LIN {X 0,Y 62.695,Z 614.162,A -85,B 0,C 180,E1 -28667.729,E2 -28667.729} C_VEL
LIN {X 0,Y 62.128,Z 611.496,A -85,B 0,C 180,E1 -28675.552,E2 -28675.552} C_VEL
LIN {X 0,Y 62.961,Z 606.814,A -85,B 0,C 180,E1 -28685.536,E2 -28685.536} C_VEL
LIN {X 0,Y 64.666,Z 601.68,A -85,B 0,C 180,E1 -28693.508,E2 -28693.508} C_VEL
LIN {X 0,Y 66.583,Z 596.849,A -85,B 0,C 180,E1 -28699.352,E2 -28699.352} C_VEL
LIN {X 0,Y 69.574,Z 589.721,A -85,B 0,C 180,E1 -28705.944,E2 -28705.944} C_VEL
LIN {X 0,Y 73.049,Z 581.764,A -85,B 0,C 180,E1 -28711.375,E2 -28711.375} C_VEL
LIN {X 0,Y 74.263,Z 578.204,A -85,B 0,C 180,E1 -28713.388,E2 -28713.388} C_VEL
LIN {X 0,Y 75.02,Z 569.916,A -85,B 0,C 180,E1 -28718.075,E2 -28718.075} C_VEL
LIN {X 0,Y 75.368,Z 562.819,A -85,B 0,C 180,E1 -28721.537,E2 -28721.537} C_VEL
LIN {X 0,Y 75.411,Z 557.992,A -85,B 0,C 180,E1 -28723.736,E2 -28723.736} C_VEL
LIN {X 0,Y 75.17,Z 557.115,A -85,B 0,C 180,E1 -28724.205,E2 -28724.205} C_VEL
LIN {X 0,Y 73.982,Z 554.238,A -85,B 0,C 180,E1 -28726.014,E2 -28726.014} C_VEL
LIN {X 0,Y 71.312,Z 550.768,A -85,B 0,C 180,E1 -28729.127,E2 -28729.127} C_VEL
LIN {X 0,Y 68.058,Z 548.078,A -85,B 0,C 180,E1 -28732.584,E2 -28732.584} C_VEL
LIN {X 0,Y 63.467,Z 544.939,A -85,B 0,C 180,E1 -28737.902,E2 -28737.902} C_VEL
LIN {X 0,Y 59.445,Z 541.388,A -85,B 0,C 180,E1 -28743.729,E2 -28743.729} C_VEL
LIN {X 0,Y 58.168,Z 538.724,A -85,B 0,C 180,E1 -28746.42,E2 -28746.42} C_VEL
LIN {X 0,Y 58.056,Z 538.062,A -85,B 0,C 180,E1 -28746.892,E2 -28746.892} C_VEL
LIN {X 0,Y 58.093,Z 538.06,A -85,B 0,C 180,E1 -28756.537,E2 -28756.537} C_VEL
LIN {X 0,Y 58.073,Z 538.046,A -85,B 0,C 180,E1 -28762.763,E2 -28762.763} C_VEL
LIN {X 0,Y 58.154,Z 538.049,A -85,B 0,C 180,E1 -28771.091,E2 -28771.091} C_VEL
LIN {X 0,Y 58.523,Z 538.007,A -85,B 0,C 180,E1 -28783.874,E2 -28783.874} C_VEL
LIN {X 0,Y 58.819,Z 537.971,A -85,B 0,C 180,E1 -28793.137,E2 -28793.137} C_VEL
LIN {X 0,Y 59.394,Z 537.882,A -85,B 0,C 180,E1 -28799.999,E2 -28799.999} C_VEL
LIN {X 0,Y 58.822,Z 537.967,A -85,B 0,C 180,E1 -28806.861,E2 -28806.861} C_VEL
LIN {X 0,Y 58.656,Z 537.992,A -85,B 0,C 180,E1 -28813.864,E2 -28813.864} C_VEL
LIN {X 0,Y 58.313,Z 538.113,A -85,B 0,C 180,E1 -28819.168,E2 -28819.168} C_VEL
LIN {X 0,Y 59.17,Z 540.867,A -85,B 0,C 180,E1 -28821.33,E2 -28821.33} C_VEL
LIN {X 0,Y 61.251,Z 543.062,A -85,B 0,C 180,E1 -28824.578,E2 -28824.578} C_VEL
LIN {X 0,Y 63.526,Z 546.992,A -85,B 0,C 180,E1 -28828.49,E2 -28828.49} C_VEL
LIN {X 0,Y 65.839,Z 551.416,A -85,B 0,C 180,E1 -28832.257,E2 -28832.257} C_VEL
LIN {X 0,Y 67.801,Z 556.21,A -85,B 0,C 180,E1 -28835.78,E2 -28835.78} C_VEL
LIN {X 0,Y 69.602,Z 562.062,A -85,B 0,C 180,E1 -28839.511,E2 -28839.511} C_VEL
LIN {X 0,Y 69.534,Z 564.952,A -85,B 0,C 180,E1 -28840.948,E2 -28840.948} C_VEL
LIN {X 0,Y 68.595,Z 571.827,A -85,B 0,C 180,E1 -28844.181,E2 -28844.181} C_VEL
LIN {X 0,Y 67.006,Z 579.314,A -85,B 0,C 180,E1 -28848.237,E2 -28848.237} C_VEL
LIN {X 0,Y 65.019,Z 587.202,A -85,B 0,C 180,E1 -28853.527,E2 -28853.527} C_VEL
LIN {X 0,Y 61.812,Z 594.337,A -85,B 0,C 180,E1 -28859.23,E2 -28859.23} C_VEL
LIN {X 0,Y 58.654,Z 601.567,A -85,B 0,C 180,E1 -28867.086,E2 -28867.086} C_VEL
LIN {X 0,Y 56.668,Z 607.224,A -85,B 0,C 180,E1 -28875.642,E2 -28875.642} C_VEL
LIN {X 0,Y 55.889,Z 610.89,A -85,B 0,C 180,E1 -28882.78,E2 -28882.78} C_VEL
LIN {X 0,Y 55.823,Z 613.824,A -85,B 0,C 180,E1 -28890.004,E2 -28890.004} C_VEL
LIN {X 0,Y 55.911,Z 616.058,A -85,B 0,C 180,E1 -28897.225,E2 -28897.225} C_VEL
LIN {X 0,Y 56.666,Z 617.777,A -85,B 0,C 180,E1 -28904.366,E2 -28904.366} C_VEL
LIN {X 0,Y 58.234,Z 619.04,A -85,B 0,C 180,E1 -28911.23,E2 -28911.23} C_VEL
LIN {X 0,Y 60.598,Z 619.853,A -85,B 0,C 180,E1 -28917.644,E2 -28917.644} C_VEL
LIN {X 0,Y 63.711,Z 620.113,A -85,B 0,C 180,E1 -28923.477,E2 -28923.477} C_VEL
LIN {X 0,Y 67.391,Z 619.924,A -85,B 0,C 180,E1 -28928.739,E2 -28928.739} C_VEL
LIN {X 0,Y 71.697,Z 619.325,A -85,B 0,C 180,E1 -28933.331,E2 -28933.331} C_VEL
LIN {X 0,Y 78.242,Z 617.748,A -85,B 0,C 180,E1 -28938.535,E2 -28938.535} C_VEL
LIN {X 0,Y 79.106,Z 617.273,A -85,B 0,C 180,E1 -28940.327,E2 -28940.327} C_VEL
LIN {X 0,Y 70.642,Z 617.379,A -85,B 0,C 180,E1 -28953.565,E2 -28953.565} C_VEL
LIN {X 0,Y 68.291,Z 617.214,A -85,B 0,C 180,E1 -28974.094,E2 -28974.094} C_VEL
LIN {X 0,Y 73.617,Z 616.962,A -85,B 0,C 180,E1 -28991.008,E2 -28991.008} C_VEL
LIN {X 0,Y 72.382,Z 617.292,A -85,B 0,C 180,E1 -28993.831,E2 -28993.831} C_VEL
LIN {X 0,Y 67.111,Z 617.813,A -85,B 0,C 180,E1 -28999.515,E2 -28999.515} C_VEL
LIN {X 0,Y 62.187,Z 617.57,A -85,B 0,C 180,E1 -29006.876,E2 -29006.876} C_VEL
LIN {X 0,Y 57.701,Z 616.071,A -85,B 0,C 180,E1 -29017.518,E2 -29017.518} C_VEL
LIN {X 0,Y 55.794,Z 614.098,A -85,B 0,C 180,E1 -29025.95,E2 -29025.95} C_VEL
LIN {X 0,Y 55.061,Z 611.285,A -85,B 0,C 180,E1 -29034.939,E2 -29034.939} C_VEL
LIN {X 0,Y 55.788,Z 606.887,A -85,B 0,C 180,E1 -29045.3,E2 -29045.3} C_VEL
LIN {X 0,Y 57.535,Z 601.881,A -85,B 0,C 180,E1 -29054.047,E2 -29054.047} C_VEL
LIN {X 0,Y 59.949,Z 596.175,A -85,B 0,C 180,E1 -29061.57,E2 -29061.57} C_VEL
LIN {X 0,Y 62.734,Z 589.976,A -85,B 0,C 180,E1 -29067.78,E2 -29067.78} C_VEL
LIN {X 0,Y 66.583,Z 581.828,A -85,B 0,C 180,E1 -29073.78,E2 -29073.78} C_VEL
LIN {X 0,Y 67.622,Z 579.433,A -85,B 0,C 180,E1 -29075.215,E2 -29075.215} C_VEL
LIN {X 0,Y 68.657,Z 571.318,A -85,B 0,C 180,E1 -29080.316,E2 -29080.316} C_VEL
LIN {X 0,Y 69.33,Z 562.621,A -85,B 0,C 180,E1 -29084.967,E2 -29084.967} C_VEL
LIN {X 0,Y 69.031,Z 558.853,A -85,B 0,C 180,E1 -29087.144,E2 -29087.144} C_VEL
LIN {X 0,Y 67.966,Z 555.579,A -85,B 0,C 180,E1 -29089.341,E2 -29089.341} C_VEL
LIN {X 0,Y 64.392,Z 548.919,A -85,B 0,C 180,E1 -29095.202,E2 -29095.202} C_VEL
LIN {X 0,Y 63.008,Z 546.562,A -85,B 0,C 180,E1 -29097.472,E2 -29097.472} C_VEL
LIN {X 0,Y 61.362,Z 543.342,A -85,B 0,C 180,E1 -29100.642,E2 -29100.642} C_VEL
LIN {X 0,Y 59.445,Z 541.388,A -85,B 0,C 180,E1 -29103.729,E2 -29103.729} C_VEL
LIN {X 0,Y 57.754,Z 539.849,A -85,B 0,C 180,E1 -29106.813,E2 -29106.813} C_VEL
LIN {X 0,Y 55.365,Z 538.798,A -85,B 0,C 180,E1 -29112.164,E2 -29112.164} C_VEL
LIN {X 0,Y 51.647,Z 538.859,A -85,B 0,C 180,E1 -29126.839,E2 -29126.839} C_VEL
LIN {X 0,Y 51.022,Z 538.937,A -85,B 0,C 180,E1 -29135.976,E2 -29135.976} C_VEL
LIN {X 0,Y 51.464,Z 538.886,A -85,B 0,C 180,E1 -29144.149,E2 -29144.149} C_VEL
LIN {X 0,Y 51.693,Z 538.858,A -85,B 0,C 180,E1 -29152.185,E2 -29152.185} C_VEL
LIN {X 0,Y 52.278,Z 538.768,A -85,B 0,C 180,E1 -29159.999,E2 -29159.999} C_VEL
LIN {X 0,Y 51.764,Z 538.916,A -85,B 0,C 180,E1 -29167.067,E2 -29167.067} C_VEL
LIN {X 0,Y 52.378,Z 541.324,A -85,B 0,C 180,E1 -29169.899,E2 -29169.899} C_VEL
LIN {X 0,Y 54.551,Z 543.862,A -85,B 0,C 180,E1 -29175.523,E2 -29175.523} C_VEL
LIN {X 0,Y 55.092,Z 545.09,A -85,B 0,C 180,E1 -29177.132,E2 -29177.132} C_VEL
LIN {X 0,Y 56.777,Z 548.148,A -85,B 0,C 180,E1 -29181.324,E2 -29181.324} C_VEL
LIN {X 0,Y 57.757,Z 549.545,A -85,B 0,C 180,E1 -29183.294,E2 -29183.294} C_VEL
LIN {X 0,Y 60.011,Z 553.818,A -85,B 0,C 180,E1 -29187.933,E2 -29187.933} C_VEL
LIN {X 0,Y 62.036,Z 558.876,A -85,B 0,C 180,E1 -29192.556,E2 -29192.556} C_VEL
LIN {X 0,Y 63.709,Z 565.118,A -85,B 0,C 180,E1 -29197.357,E2 -29197.357} C_VEL
LIN {X 0,Y 62.218,Z 573.636,A -85,B 0,C 180,E1 -29201.785,E2 -29201.785} C_VEL
LIN {X 0,Y 59.828,Z 582.818,A -85,B 0,C 180,E1 -29207.515,E2 -29207.515} C_VEL
LIN {X 0,Y 58.504,Z 587.143,A -85,B 0,C 180,E1 -29210.905,E2 -29210.905} C_VEL
LIN {X 0,Y 55.032,Z 594.238,A -85,B 0,C 180,E1 -29217.133,E2 -29217.133} C_VEL
LIN {X 0,Y 51.604,Z 601.423,A -85,B 0,C 180,E1 -29225.889,E2 -29225.889} C_VEL
LIN {X 0,Y 49.842,Z 606.04,A -85,B 0,C 180,E1 -29233.624,E2 -29233.624} C_VEL
LIN {X 0,Y 48.721,Z 611.455,A -85,B 0,C 180,E1 -29245.868,E2 -29245.868} C_VEL
LIN {X 0,Y 48.752,Z 614.253,A -85,B 0,C 180,E1 -29254.138,E2 -29254.138} C_VEL
LIN {X 0,Y 49.84,Z 617.198,A -85,B 0,C 180,E1 -29266.385,E2 -29266.385} C_VEL
LIN {X 0,Y 51.675,Z 618.606,A -85,B 0,C 180,E1 -29274.084,E2 -29274.084} C_VEL
LIN {X 0,Y 54.402,Z 619.453,A -85,B 0,C 180,E1 -29281.119,E2 -29281.119} C_VEL
LIN {X 0,Y 57.907,Z 619.839,A -85,B 0,C 180,E1 -29287.366,E2 -29287.366} C_VEL
LIN {X 0,Y 62.004,Z 619.815,A -85,B 0,C 180,E1 -29292.855,E2 -29292.855} C_VEL
LIN {X 0,Y 68.75,Z 618.99,A -85,B 0,C 180,E1 -29299.159,E2 -29299.159} C_VEL
LIN {X 0,Y 69.788,Z 618.793,A -85,B 0,C 180,E1 -29299.946,E2 -29299.946} C_VEL
LIN {X 0,Y 69.165,Z 618.619,A -85,B 0,C 180,E1 -29302.435,E2 -29302.435} C_VEL
LIN {X 0,Y 63.323,Z 618.493,A -85,B 0,C 180,E1 -29313.645,E2 -29313.645} C_VEL
LIN {X 0,Y 64.036,Z 617.969,A -85,B 0,C 180,E1 -29346.301,E2 -29346.301} C_VEL
LIN {X 0,Y 64.716,Z 617.917,A -85,B 0,C 180,E1 -29352.196,E2 -29352.196} C_VEL
LIN {X 0,Y 57.108,Z 617.782,A -85,B 0,C 180,E1 -29361.666,E2 -29361.666} C_VEL
LIN {X 0,Y 51.18,Z 615.982,A -85,B 0,C 180,E1 -29374.514,E2 -29374.514} C_VEL
LIN {X 0,Y 48.583,Z 613.246,A -85,B 0,C 180,E1 -29386.329,E2 -29386.329} C_VEL
LIN {X 0,Y 48.028,Z 609.647,A -85,B 0,C 180,E1 -29397.94,E2 -29397.94} C_VEL
LIN {X 0,Y 49.234,Z 605.023,A -85,B 0,C 180,E1 -29409.088,E2 -29409.088} C_VEL
LIN {X 0,Y 51.955,Z 598.515,A -85,B 0,C 180,E1 -29420.364,E2 -29420.364} C_VEL
LIN {X 0,Y 55.061,Z 592.098,A -85,B 0,C 180,E1 -29428.168,E2 -29428.168} C_VEL
LIN {X 0,Y 59.108,Z 584.086,A -85,B 0,C 180,E1 -29435.113,E2 -29435.113} C_VEL
LIN {X 0,Y 61.302,Z 579.472,A -85,B 0,C 180,E1 -29438.236,E2 -29438.236} C_VEL
LIN {X 0,Y 62.604,Z 571.117,A -85,B 0,C 180,E1 -29443.936,E2 -29443.936} C_VEL
LIN {X 0,Y 63.382,Z 564.173,A -85,B 0,C 180,E1 -29448.03,E2 -29448.03} C_VEL
LIN {X 0,Y 63.056,Z 561.043,A -85,B 0,C 180,E1 -29450.147,E2 -29450.147} C_VEL
LIN {X 0,Y 61.446,Z 557.149,A -85,B 0,C 180,E1 -29453.791,E2 -29453.791} C_VEL
LIN {X 0,Y 58.569,Z 551.505,A -85,B 0,C 180,E1 -29459.958,E2 -29459.958} C_VEL
LIN {X 0,Y 56.666,Z 548.126,A -85,B 0,C 180,E1 -29464.119,E2 -29464.119} C_VEL
LIN {X 0,Y 54.868,Z 545.195,A -85,B 0,C 180,E1 -29468.459,E2 -29468.459} C_VEL
LIN {X 0,Y 54.606,Z 544.308,A -85,B 0,C 180,E1 -29469.445,E2 -29469.445} C_VEL
LIN {X 0,Y 52.065,Z 541.823,A -85,B 0,C 180,E1 -29476.147,E2 -29476.147} C_VEL
LIN {X 0,Y 51.012,Z 539.312,A -85,B 0,C 180,E1 -29480.336,E2 -29480.336} C_VEL
LIN {X 0,Y 50.965,Z 538.935,A -85,B 0,C 180,E1 -29480.918,E2 -29480.918} C_VEL
LIN {X 0,Y 51.072,Z 538.928,A -85,B 0,C 180,E1 -29486.602,E2 -29486.602} C_VEL
LIN {X 0,Y 51.022,Z 538.937,A -85,B 0,C 180,E1 -29495.976,E2 -29495.976} C_VEL
LIN {X 0,Y 50.829,Z 539.191,A -85,B 0,C 180,E1 -29500.356,E2 -29500.356} C_VEL
LIN {X 0,Y 50.155,Z 540.411,A -85,B 0,C 180,E1 -29506.853,E2 -29506.853} C_VEL
LIN {X 0,Y 49.075,Z 543.87,A -85,B 0,C 180,E1 -29517.658,E2 -29517.658} C_VEL
LIN {X 0,Y 50.332,Z 548.838,A -85,B 0,C 180,E1 -29530.483,E2 -29530.483} C_VEL
LIN {X 0,Y 51.408,Z 550.333,A -85,B 0,C 180,E1 -29533.841,E2 -29533.841} C_VEL
LIN {X 0,Y 54.282,Z 556.387,A -85,B 0,C 180,E1 -29542.855,E2 -29542.855} C_VEL
LIN {X 0,Y 56.192,Z 560.773,A -85,B 0,C 180,E1 -29547.97,E2 -29547.97} C_VEL
LIN {X 0,Y 57.562,Z 566.47,A -85,B 0,C 180,E1 -29553.323,E2 -29553.323} C_VEL
LIN {X 0,Y 57.709,Z 567.701,A -85,B 0,C 180,E1 -29554.277,E2 -29554.277} C_VEL
LIN {X 0,Y 55.801,Z 575.775,A -85,B 0,C 180,E1 -29559.03,E2 -29559.03} C_VEL
LIN {X 0,Y 52.873,Z 584.913,A -85,B 0,C 180,E1 -29565.751,E2 -29565.751} C_VEL
LIN {X 0,Y 52.129,Z 587.007,A -85,B 0,C 180,E1 -29567.622,E2 -29567.622} C_VEL
LIN {X 0,Y 48.349,Z 594.094,A -85,B 0,C 180,E1 -29574.453,E2 -29574.453} C_VEL
LIN {X 0,Y 44.608,Z 601.265,A -85,B 0,C 180,E1 -29584.33,E2 -29584.33} C_VEL
LIN {X 0,Y 42.359,Z 606.876,A -85,B 0,C 180,E1 -29595.594,E2 -29595.594} C_VEL
LIN {X 0,Y 41.688,Z 610.528,A -85,B 0,C 180,E1 -29605.17,E2 -29605.17} C_VEL
LIN {X 0,Y 41.735,Z 613.407,A -85,B 0,C 180,E1 -29614.835,E2 -29614.835} C_VEL
LIN {X 0,Y 43.1,Z 616.595,A -85,B 0,C 180,E1 -29629.039,E2 -29629.039} C_VEL
LIN {X 0,Y 45.29,Z 618.046,A -85,B 0,C 180,E1 -29637.75,E2 -29637.75} C_VEL
LIN {X 0,Y 48.458,Z 619.012,A -85,B 0,C 180,E1 -29645.465,E2 -29645.465} C_VEL
LIN {X 0,Y 52.429,Z 619.564,A -85,B 0,C 180,E1 -29652.091,E2 -29652.091} C_VEL
LIN {X 0,Y 59.289,Z 619.538,A -85,B 0,C 180,E1 -29659.922,E2 -29659.922} C_VEL
LIN {X 0,Y 60.468,Z 619.454,A -85,B 0,C 180,E1 -29660.957,E2 -29660.957} C_VEL
LIN {X 0,Y 59.941,Z 619.329,A -85,B 0,C 180,E1 -29664.11,E2 -29664.11} C_VEL
LIN {X 0,Y 53.968,Z 618.847,A -85,B 0,C 180,E1 -29684.904,E2 -29684.904} C_VEL
LIN {X 0,Y 56.855,Z 618.349,A -85,B 0,C 180,E1 -29707.101,E2 -29707.101} C_VEL
LIN {X 0,Y 57.117,Z 618.308,A -85,B 0,C 180,E1 -29710.123,E2 -29710.123} C_VEL
LIN {X 0,Y 51.48,Z 617.892,A -85,B 0,C 180,E1 -29717.118,E2 -29717.118} C_VEL
LIN {X 0,Y 46.088,Z 616.519,A -85,B 0,C 180,E1 -29727.225,E2 -29727.225} C_VEL
LIN {X 0,Y 42.027,Z 613.504,A -85,B 0,C 180,E1 -29741.984,E2 -29741.984} C_VEL
LIN {X 0,Y 40.982,Z 608.87,A -85,B 0,C 180,E1 -29759.032,E2 -29759.032} C_VEL
LIN {X 0,Y 42.883,Z 603.048,A -85,B 0,C 180,E1 -29773.865,E2 -29773.865} C_VEL
LIN {X 0,Y 45.356,Z 597.831,A -85,B 0,C 180,E1 -29783.322,E2 -29783.322} C_VEL
LIN {X 0,Y 49.25,Z 590.567,A -85,B 0,C 180,E1 -29792.669,E2 -29792.669} C_VEL
LIN {X 0,Y 53.459,Z 582.912,A -85,B 0,C 180,E1 -29799.455,E2 -29799.455} C_VEL
LIN {X 0,Y 55.139,Z 579.414,A -85,B 0,C 180,E1 -29801.95,E2 -29801.95} C_VEL
LIN {X 0,Y 56.756,Z 571.197,A -85,B 0,C 180,E1 -29808.085,E2 -29808.085} C_VEL
LIN {X 0,Y 57.596,Z 566.097,A -85,B 0,C 180,E1 -29811.47,E2 -29811.47} C_VEL
LIN {X 0,Y 57.5,Z 564.645,A -85,B 0,C 180,E1 -29812.567,E2 -29812.567} C_VEL
LIN {X 0,Y 55.027,Z 558.471,A -85,B 0,C 180,E1 -29819.75,E2 -29819.75} C_VEL
LIN {X 0,Y 52.596,Z 553.489,A -85,B 0,C 180,E1 -29826.702,E2 -29826.702} C_VEL
LIN {X 0,Y 51.361,Z 551.013,A -85,B 0,C 180,E1 -29830.958,E2 -29830.958} C_VEL
LIN {X 0,Y 48.553,Z 546.463,A -85,B 0,C 180,E1 -29841.704,E2 -29841.704} C_VEL
LIN {X 0,Y 48.349,Z 545.497,A -85,B 0,C 180,E1 -29843.47,E2 -29843.47} C_VEL
LIN {X 0,Y 46.285,Z 543.916,A -85,B 0,C 180,E1 -29862.32,E2 -29862.32} C_VEL
LIN {X 0,Y 47.355,Z 544.32,A -85,B 0,C 180,E1 -29875.744,E2 -29875.744} C_VEL
LIN {X 0,Y 48.507,Z 544.918,A -85,B 0,C 180,E1 -29881.712,E2 -29881.712} C_VEL
LIN {X 0,Y 49.051,Z 545.56,A -85,B 0,C 180,E1 -29884.236,E2 -29884.236} C_VEL
LIN {X 0,Y 50.002,Z 548.374,A -85,B 0,C 180,E1 -29889.352,E2 -29889.352} C_VEL
LIN {X 0,Y 50.332,Z 548.838,A -85,B 0,C 180,E1 -29890.483,E2 -29890.483} C_VEL
LIN {X 0,Y 51.221,Z 551.05,A -85,B 0,C 180,E1 -29893.942,E2 -29893.942} C_VEL
LIN {X 0,Y 51.425,Z 554.113,A -85,B 0,C 180,E1 -29896.75,E2 -29896.75} C_VEL
LIN {X 0,Y 50.92,Z 563.332,A -85,B 0,C 180,E1 -29903.585,E2 -29903.585} C_VEL
LIN {X 0,Y 51.151,Z 565.347,A -85,B 0,C 180,E1 -29905.697,E2 -29905.697} C_VEL
LIN {X 0,Y 51.921,Z 569.636,A -85,B 0,C 180,E1 -29910.268,E2 -29910.268} C_VEL
LIN {X 0,Y 49.605,Z 577.426,A -85,B 0,C 180,E1 -29915.454,E2 -29915.454} C_VEL
LIN {X 0,Y 46.4,Z 585.8,A -85,B 0,C 180,E1 -29922.411,E2 -29922.411} C_VEL
LIN {X 0,Y 43.791,Z 590.622,A -85,B 0,C 180,E1 -29927.001,E2 -29927.001} C_VEL
LIN {X 0,Y 39.965,Z 596.971,A -85,B 0,C 180,E1 -29935.15,E2 -29935.15} C_VEL
LIN {X 0,Y 36.497,Z 603.391,A -85,B 0,C 180,E1 -29947.354,E2 -29947.354} C_VEL
LIN {X 0,Y 34.97,Z 607.581,A -85,B 0,C 180,E1 -29958.412,E2 -29958.412} C_VEL
LIN {X 0,Y 34.657,Z 611.036,A -85,B 0,C 180,E1 -29970.006,E2 -29970.006} C_VEL
LIN {X 0,Y 35.041,Z 613.784,A -85,B 0,C 180,E1 -29981.576,E2 -29981.576} C_VEL
LIN {X 0,Y 36.493,Z 615.875,A -85,B 0,C 180,E1 -29992.66,E2 -29992.66} C_VEL
LIN {X 0,Y 39.155,Z 617.439,A -85,B 0,C 180,E1 -30002.586,E2 -30002.586} C_VEL
LIN {X 0,Y 42.871,Z 618.571,A -85,B 0,C 180,E1 -30010.981,E2 -30010.981} C_VEL
LIN {X 0,Y 49.877,Z 619.402,A -85,B 0,C 180,E1 -30020.809,E2 -30020.809} C_VEL
LIN {X 0,Y 51.17,Z 619.46,A -85,B 0,C 180,E1 -30022.167,E2 -30022.167} C_VEL
LIN {X 0,Y 51.448,Z 619.447,A -85,B 0,C 180,E1 -30025.054,E2 -30025.054} C_VEL
LIN {X 0,Y 47.728,Z 618.464,A -85,B 0,C 180,E1 -30060.001,E2 -30060.001} C_VEL
LIN {X 0,Y 48.79,Z 618.197,A -85,B 0,C 180,E1 -30068.283,E2 -30068.283} C_VEL
LIN {X 0,Y 41.074,Z 616.73,A -85,B 0,C 180,E1 -30080.012,E2 -30080.012} C_VEL
LIN {X 0,Y 35.753,Z 613.724,A -85,B 0,C 180,E1 -30096.138,E2 -30096.138} C_VEL
LIN {X 0,Y 33.905,Z 610.286,A -85,B 0,C 180,E1 -30111.541,E2 -30111.541} C_VEL
LIN {X 0,Y 34.784,Z 605.274,A -85,B 0,C 180,E1 -30128.967,E2 -30128.967} C_VEL
LIN {X 0,Y 38.098,Z 598.596,A -85,B 0,C 180,E1 -30144.702,E2 -30144.702} C_VEL
LIN {X 0,Y 41.274,Z 593.25,A -85,B 0,C 180,E1 -30153.268,E2 -30153.268} C_VEL
LIN {X 0,Y 46.195,Z 585.066,A -85,B 0,C 180,E1 -30162.07,E2 -30162.07} C_VEL
LIN {X 0,Y 48.907,Z 580.507,A -85,B 0,C 180,E1 -30165.627,E2 -30165.627} C_VEL
LIN {X 0,Y 51,Z 572.463,A -85,B 0,C 180,E1 -30172.265,E2 -30172.265} C_VEL
LIN {X 0,Y 51.88,Z 567.997,A -85,B 0,C 180,E1 -30175.604,E2 -30175.604} C_VEL
LIN {X 0,Y 50.077,Z 562.836,A -85,B 0,C 180,E1 -30182.64,E2 -30182.64} C_VEL
LIN {X 0,Y 48.963,Z 559.738,A -85,B 0,C 180,E1 -30187.611,E2 -30187.611} C_VEL
LIN {X 0,Y 47.774,Z 557.116,A -85,B 0,C 180,E1 -30192.646,E2 -30192.646} C_VEL
LIN {X 0,Y 45.881,Z 553.487,A -85,B 0,C 180,E1 -30202.213,E2 -30202.213} C_VEL
LIN {X 0,Y 44.71,Z 551.511,A -85,B 0,C 180,E1 -30211.863,E2 -30211.863} C_VEL
LIN {X 0,Y 44.204,Z 550.713,A -85,B 0,C 180,E1 -30222.529,E2 -30222.529} C_VEL
LIN {X 0,Y 44.638,Z 550.808,A -85,B 0,C 180,E1 -30230.941,E2 -30230.941} C_VEL
LIN {X 0,Y 45.985,Z 551.42,A -85,B 0,C 180,E1 -30239.999,E2 -30239.999} C_VEL
LIN {X 0,Y 47.813,Z 556.397,A -85,B 0,C 180,E1 -30251.687,E2 -30251.687} C_VEL
LIN {X 0,Y 49.951,Z 561.613,A -85,B 0,C 180,E1 -30260.593,E2 -30260.593} C_VEL
LIN {X 0,Y 51.151,Z 565.347,A -85,B 0,C 180,E1 -30265.697,E2 -30265.697} C_VEL
LIN {X 0,Y 51.217,Z 567.366,A -85,B 0,C 180,E1 -30267.476,E2 -30267.476} C_VEL
LIN {X 0,Y 50.006,Z 570.782,A -85,B 0,C 180,E1 -30269.219,E2 -30269.219} C_VEL
LIN {X 0,Y 47.99,Z 574.091,A -85,B 0,C 180,E1 -30270.317,E2 -30270.317} C_VEL
LIN {X 0,Y 43.031,Z 580.89,A -85,B 0,C 180,E1 -30272.782,E2 -30272.782} C_VEL
LIN {X 0,Y 41.805,Z 583.132,A -85,B 0,C 180,E1 -30274.468,E2 -30274.468} C_VEL
LIN {X 0,Y 40.149,Z 586.581,A -85,B 0,C 180,E1 -30278.036,E2 -30278.036} C_VEL
LIN {X 0,Y 35.46,Z 593.648,A -85,B 0,C 180,E1 -30286.086,E2 -30286.086} C_VEL
LIN {X 0,Y 30.78,Z 600.81,A -85,B 0,C 180,E1 -30299.094,E2 -30299.094} C_VEL
LIN {X 0,Y 28.069,Z 606.416,A -85,B 0,C 180,E1 -30315.507,E2 -30315.507} C_VEL
LIN {X 0,Y 27.619,Z 610.053,A -85,B 0,C 180,E1 -30330.007,E2 -30330.007} C_VEL
LIN {X 0,Y 28.952,Z 614.052,A -85,B 0,C 180,E1 -30351.361,E2 -30351.361} C_VEL
LIN {X 0,Y 33.405,Z 616.813,A -85,B 0,C 180,E1 -30369.144,E2 -30369.144} C_VEL
LIN {X 0,Y 37.8,Z 618.115,A -85,B 0,C 180,E1 -30378.055,E2 -30378.055} C_VEL
LIN {X 0,Y 42.943,Z 618.94,A -85,B 0,C 180,E1 -30384.922,E2 -30384.922} C_VEL
LIN {X 0,Y 42.089,Z 618.862,A -85,B 0,C 180,E1 -30389.939,E2 -30389.939} C_VEL
LIN {X 0,Y 40.517,Z 617.965,A -85,B 0,C 180,E1 -30420.001,E2 -30420.001} C_VEL
LIN {X 0,Y 41.069,Z 617.773,A -85,B 0,C 180,E1 -30424.909,E2 -30424.909} C_VEL
LIN {X 0,Y 35.999,Z 616.637,A -85,B 0,C 180,E1 -30432.516,E2 -30432.516} C_VEL
LIN {X 0,Y 30.036,Z 613.939,A -85,B 0,C 180,E1 -30447.904,E2 -30447.904} C_VEL
LIN {X 0,Y 27.076,Z 610.432,A -85,B 0,C 180,E1 -30466.624,E2 -30466.624} C_VEL
LIN {X 0,Y 27.393,Z 605.744,A -85,B 0,C 180,E1 -30487.358,E2 -30487.358} C_VEL
LIN {X 0,Y 30.855,Z 599.295,A -85,B 0,C 180,E1 -30506.729,E2 -30506.729} C_VEL
LIN {X 0,Y 35.651,Z 592.034,A -85,B 0,C 180,E1 -30519.707,E2 -30519.707} C_VEL
LIN {X 0,Y 40.5,Z 584.856,A -85,B 0,C 180,E1 -30527.674,E2 -30527.674} C_VEL
LIN {X 0,Y 43.351,Z 580.298,A -85,B 0,C 180,E1 -30531.388,E2 -30531.388} C_VEL
LIN {X 0,Y 46.102,Z 571.554,A -85,B 0,C 180,E1 -30539.099,E2 -30539.099} C_VEL
LIN {X 0,Y 45.844,Z 569.564,A -85,B 0,C 180,E1 -30541.899,E2 -30541.899} C_VEL
LIN {X 0,Y 44.386,Z 564.472,A -85,B 0,C 180,E1 -30551.219,E2 -30551.219} C_VEL
LIN {X 0,Y 43.199,Z 561.16,A -85,B 0,C 180,E1 -30559.401,E2 -30559.401} C_VEL
LIN {X 0,Y 42.515,Z 559.364,A -85,B 0,C 180,E1 -30565.735,E2 -30565.735} C_VEL
LIN {X 0,Y 42.102,Z 558.587,A -85,B 0,C 180,E1 -30569.947,E2 -30569.947} C_VEL
LIN {X 0,Y 41.586,Z 557.515,A -85,B 0,C 180,E1 -30580.244,E2 -30580.244} C_VEL
LIN {X 0,Y 41.994,Z 557.396,A -85,B 0,C 180,E1 -30590.365,E2 -30590.365} C_VEL
LIN {X 0,Y 42.384,Z 557.622,A -85,B 0,C 180,E1 -30594.171,E2 -30594.171} C_VEL
LIN {X 0,Y 43.043,Z 558.582,A -85,B 0,C 180,E1 -30599.999,E2 -30599.999} C_VEL
LIN {X 0,Y 43.994,Z 562.142,A -85,B 0,C 180,E1 -30609.192,E2 -30609.192} C_VEL
LIN {X 0,Y 45.391,Z 566.601,A -85,B 0,C 180,E1 -30618.038,E2 -30618.038} C_VEL
LIN {X 0,Y 46.044,Z 569.401,A -85,B 0,C 180,E1 -30622.436,E2 -30622.436} C_VEL
LIN {X 0,Y 46.108,Z 572.418,A -85,B 0,C 180,E1 -30626.135,E2 -30626.135} C_VEL
LIN {X 0,Y 43.566,Z 579.044,A -85,B 0,C 180,E1 -30631.017,E2 -30631.017} C_VEL
LIN {X 0,Y 41.805,Z 583.132,A -85,B 0,C 180,E1 -30634.468,E2 -30634.468} C_VEL
LIN {X 0,Y 39.809,Z 586.118,A -85,B 0,C 180,E1 -30636.673,E2 -30636.673} C_VEL
LIN {X 0,Y 36.962,Z 588.807,A -85,B 0,C 180,E1 -30637.997,E2 -30637.997} C_VEL
LIN {X 0,Y 29.388,Z 594.388,A -85,B 0,C 180,E1 -30641.359,E2 -30641.359} C_VEL
LIN {X 0,Y 26.788,Z 596.84,A -85,B 0,C 180,E1 -30645.337,E2 -30645.337} C_VEL
LIN {X 0,Y 22.481,Z 602.872,A -85,B 0,C 180,E1 -30662.045,E2 -30662.045} C_VEL
LIN {X 0,Y 20.676,Z 607.062,A -85,B 0,C 180,E1 -30680.225,E2 -30680.225} C_VEL
LIN {X 0,Y 20.787,Z 610.488,A -85,B 0,C 180,E1 -30699.743,E2 -30699.743} C_VEL
LIN {X 0,Y 22.54,Z 613.213,A -85,B 0,C 180,E1 -30717.896,E2 -30717.896} C_VEL
LIN {X 0,Y 28.27,Z 616.181,A -85,B 0,C 180,E1 -30738.24,E2 -30738.24} C_VEL
LIN {X 0,Y 33.477,Z 617.606,A -85,B 0,C 180,E1 -30747.123,E2 -30747.123} C_VEL
LIN {X 0,Y 33.649,Z 617.687,A -85,B 0,C 180,E1 -30755.31,E2 -30755.31} C_VEL
LIN {X 0,Y 33.367,Z 617.021,A -85,B 0,C 180,E1 -30780.001,E2 -30780.001} C_VEL
LIN {X 0,Y 28.422,Z 615.52,A -85,B 0,C 180,E1 -30788.423,E2 -30788.423} C_VEL
LIN {X 0,Y 23.025,Z 612.907,A -85,B 0,C 180,E1 -30803.671,E2 -30803.671} C_VEL
LIN {X 0,Y 19.753,Z 608.532,A -85,B 0,C 180,E1 -30831.477,E2 -30831.477} C_VEL
LIN {X 0,Y 21.478,Z 603.062,A -85,B 0,C 180,E1 -30859.011,E2 -30859.011} C_VEL
LIN {X 0,Y 24.743,Z 598.427,A -85,B 0,C 180,E1 -30874.064,E2 -30874.064} C_VEL
LIN {X 0,Y 30.238,Z 591.351,A -85,B 0,C 180,E1 -30887.628,E2 -30887.628} C_VEL
LIN {X 0,Y 35.308,Z 584.647,A -85,B 0,C 180,E1 -30895.017,E2 -30895.017} C_VEL
LIN {X 0,Y 37.782,Z 581.245,A -85,B 0,C 180,E1 -30897.706,E2 -30897.706} C_VEL
LIN {X 0,Y 40.488,Z 574.907,A -85,B 0,C 180,E1 -30903.839,E2 -30903.839} C_VEL
LIN {X 0,Y 40.598,Z 573.268,A -85,B 0,C 180,E1 -30906.26,E2 -30906.26} C_VEL
LIN {X 0,Y 39.864,Z 569.193,A -85,B 0,C 180,E1 -30915.153,E2 -30915.153} C_VEL
LIN {X 0,Y 39.351,Z 566.719,A -85,B 0,C 180,E1 -30922.534,E2 -30922.534} C_VEL
LIN {X 0,Y 39.032,Z 565.512,A -85,B 0,C 180,E1 -30927.304,E2 -30927.304} C_VEL
LIN {X 0,Y 38.521,Z 564.132,A -85,B 0,C 180,E1 -30938.598,E2 -30938.598} C_VEL
LIN {X 0,Y 38.9,Z 563.834,A -85,B 0,C 180,E1 -30949.59,E2 -30949.59} C_VEL
LIN {X 0,Y 39.638,Z 565.348,A -85,B 0,C 180,E1 -30959.999,E2 -30959.999} C_VEL
LIN {X 0,Y 40.227,Z 569.153,A -85,B 0,C 180,E1 -30970.061,E2 -30970.061} C_VEL
LIN {X 0,Y 40.823,Z 572.671,A -85,B 0,C 180,E1 -30977.533,E2 -30977.533} C_VEL
LIN {X 0,Y 40.879,Z 574.327,A -85,B 0,C 180,E1 -30980.11,E2 -30980.11} C_VEL
LIN {X 0,Y 35.995,Z 584.207,A -85,B 0,C 180,E1 -30988.536,E2 -30988.536} C_VEL
LIN {X 0,Y 33.432,Z 588.281,A -85,B 0,C 180,E1 -30992.778,E2 -30992.778} C_VEL
LIN {X 0,Y 26.788,Z 596.84,A -85,B 0,C 180,E1 -31005.337,E2 -31005.337} C_VEL
LIN {X 0,Y 23.543,Z 600.418,A -85,B 0,C 180,E1 -31013.444,E2 -31013.444} C_VEL
LIN {X 0,Y 19.981,Z 603.466,A -85,B 0,C 180,E1 -31023.106,E2 -31023.106} C_VEL
LIN {X 0,Y 14.656,Z 608.552,A -85,B 0,C 180,E1 -31055.277,E2 -31055.277} C_VEL
LIN {X 0,Y 15.681,Z 611.492,A -85,B 0,C 180,E1 -31083.445,E2 -31083.445} C_VEL
LIN {X 0,Y 21.357,Z 614.471,A -85,B 0,C 180,E1 -31105.37,E2 -31105.37} C_VEL
LIN {X 0,Y 25.551,Z 615.877,A -85,B 0,C 180,E1 -31113.008,E2 -31113.008} C_VEL
LIN {X 0,Y 26.189,Z 616.026,A -85,B 0,C 180,E1 -31118.988,E2 -31118.988} C_VEL
LIN {X 0,Y 25.838,Z 615.721,A -85,B 0,C 180,E1 -31132.185,E2 -31132.185} C_VEL
LIN {X 0,Y 21.095,Z 614,A -85,B 0,C 180,E1 -31141.479,E2 -31141.479} C_VEL
LIN {X 0,Y 15.138,Z 610.849,A -85,B 0,C 180,E1 -31161.758,E2 -31161.758} C_VEL
LIN {X 0,Y 12.669,Z 606.831,A -85,B 0,C 180,E1 -31196.287,E2 -31196.287} C_VEL
LIN {X 0,Y 15.346,Z 601.85,A -85,B 0,C 180,E1 -31229.987,E2 -31229.987} C_VEL
LIN {X 0,Y 20.804,Z 595.884,A -85,B 0,C 180,E1 -31249.734,E2 -31249.734} C_VEL
LIN {X 0,Y 28.243,Z 587.656,A -85,B 0,C 180,E1 -31261.915,E2 -31261.915} C_VEL
LIN {X 0,Y 33.544,Z 580.905,A -85,B 0,C 180,E1 -31267.032,E2 -31267.032} C_VEL
LIN {X 0,Y 35.139,Z 577.71,A -85,B 0,C 180,E1 -31270.278,E2 -31270.278} C_VEL
LIN {X 0,Y 35.419,Z 576.114,A -85,B 0,C 180,E1 -31273.441,E2 -31273.441} C_VEL
LIN {X 0,Y 35.312,Z 572.756,A -85,B 0,C 180,E1 -31283.338,E2 -31283.338} C_VEL
LIN {X 0,Y 35.044,Z 570.963,A -85,B 0,C 180,E1 -31293.072,E2 -31293.072} C_VEL
LIN {X 0,Y 35.01,Z 570.601,A -85,B 0,C 180,E1 -31296.328,E2 -31296.328} C_VEL
LIN {X 0,Y 35.361,Z 570.094,A -85,B 0,C 180,E1 -31308.535,E2 -31308.535} C_VEL
LIN {X 0,Y 35.453,Z 570.493,A -85,B 0,C 180,E1 -31312.339,E2 -31312.339} C_VEL
LIN {X 0,Y 35.711,Z 571.893,A -85,B 0,C 180,E1 -31319.999,E2 -31319.999} C_VEL
LIN {X 0,Y 35.813,Z 575.999,A -85,B 0,C 180,E1 -31331.316,E2 -31331.316} C_VEL
LIN {X 0,Y 35.404,Z 577.398,A -85,B 0,C 180,E1 -31333.539,E2 -31333.539} C_VEL
LIN {X 0,Y 30.868,Z 584.858,A -85,B 0,C 180,E1 -31340.107,E2 -31340.107} C_VEL
LIN {X 0,Y 27.102,Z 589.735,A -85,B 0,C 180,E1 -31344.843,E2 -31344.843} C_VEL
LIN {X 0,Y 20.04,Z 597.478,A -85,B 0,C 180,E1 -31357.917,E2 -31357.917} C_VEL
LIN {X 0,Y 14.866,Z 603.671,A -85,B 0,C 180,E1 -31381.803,E2 -31381.803} C_VEL
LIN {X 0,Y 13.55,Z 607.665,A -85,B 0,C 180,E1 -31410.015,E2 -31410.015} C_VEL
LIN {X 0,Y 15.007,Z 610.868,A -85,B 0,C 180,E1 -31437.94,E2 -31437.94} C_VEL
LIN {X 0,Y 15.681,Z 611.492,A -85,B 0,C 180,E1 -31443.445,E2 -31443.445} C_VEL
LIN {X 0,Y 15.584,Z 611.799,A -85,B 0,C 180,E1 -31448.466,E2 -31448.466} C_VEL
LIN {X 0,Y 14.026,Z 611.663,A -85,B 0,C 180,E1 -31456.697,E2 -31456.697} C_VEL
LIN {X 0,Y 10.524,Z 610.598,A -85,B 0,C 180,E1 -31469.876,E2 -31469.876} C_VEL
LIN {X 0,Y 7.84,Z 609.407,A -85,B 0,C 180,E1 -31482.509,E2 -31482.509} C_VEL
LIN {X 0,Y 4.639,Z 607.226,A -85,B 0,C 180,E1 -31519.052,E2 -31519.052} C_VEL
LIN {X 0,Y 6.723,Z 603.518,A -85,B 0,C 180,E1 -31595.252,E2 -31595.252} C_VEL
LIN {X 0,Y 12.291,Z 599.046,A -85,B 0,C 180,E1 -31618.997,E2 -31618.997} C_VEL
LIN {X 0,Y 19.533,Z 592.574,A -85,B 0,C 180,E1 -31630.882,E2 -31630.882} C_VEL
LIN {X 0,Y 25.675,Z 586.201,A -85,B 0,C 180,E1 -31635.922,E2 -31635.922} C_VEL
LIN {X 0,Y 29.524,Z 581.778,A -85,B 0,C 180,E1 -31637.88,E2 -31637.88} C_VEL
LIN {X 0,Y 30.23,Z 580.709,A -85,B 0,C 180,E1 -31638.719,E2 -31638.719} C_VEL
LIN {X 0,Y 30.728,Z 579.166,A -85,B 0,C 180,E1 -31642.427,E2 -31642.427} C_VEL
LIN {X 0,Y 30.908,Z 577.85,A -85,B 0,C 180,E1 -31647.961,E2 -31647.961} C_VEL
LIN {X 0,Y 31.031,Z 576.77,A -85,B 0,C 180,E1 -31654.934,E2 -31654.934} C_VEL
LIN {X 0,Y 31.377,Z 576.161,A -85,B 0,C 180,E1 -31667.056,E2 -31667.056} C_VEL
LIN {X 0,Y 31.47,Z 576.436,A -85,B 0,C 180,E1 -31671.362,E2 -31671.362} C_VEL
LIN {X 0,Y 31.213,Z 578.254,A -85,B 0,C 180,E1 -31679.999,E2 -31679.999} C_VEL
LIN {X 0,Y 31.073,Z 579.147,A -85,B 0,C 180,E1 -31683.082,E2 -31683.082} C_VEL
LIN {X 0,Y 29.206,Z 582.169,A -85,B 0,C 180,E1 -31685.829,E2 -31685.829} C_VEL
LIN {X 0,Y 26.66,Z 585.496,A -85,B 0,C 180,E1 -31688.729,E2 -31688.729} C_VEL
LIN {X 0,Y 21.598,Z 590.999,A -85,B 0,C 180,E1 -31692.564,E2 -31692.564} C_VEL
LIN {X 0,Y 15.067,Z 597.131,A -85,B 0,C 180,E1 -31701.147,E2 -31701.147} C_VEL
LIN {X 0,Y 8.123,Z 603.333,A -85,B 0,C 180,E1 -31729.576,E2 -31729.576} C_VEL
LIN {X 0,Y 6.515,Z 606.427,A -85,B 0,C 180,E1 -31770.031,E2 -31770.031} C_VEL
LIN {X 0,Y 9.4,Z 609.829,A -85,B 0,C 180,E1 -31818.42,E2 -31818.42} C_VEL
LIN {X 0,Y 15.078,Z 612.524,A -85,B 0,C 180,E1 -31838.817,E2 -31838.817} C_VEL
LIN {X 0,Y 16.255,Z 612.94,A -85,B 0,C 180,E1 -31844.779,E2 -31844.779} C_VEL
LIN {X 0,Y 7.294,Z 608.439,A -85,B 0,C 180,E1 -31875.405,E2 -31875.405} C_VEL
LIN {X 0,Y 7.031,Z 603.621,A -85,B 0,C 180,E1 -31951.427,E2 -31951.427} C_VEL
LIN {X 0,Y 12.291,Z 599.046,A -85,B 0,C 180,E1 -31978.997,E2 -31978.997} C_VEL
LIN {X 0,Y 14.7,Z 596.634,A -85,B 0,C 180,E1 -31987.231,E2 -31987.231} C_VEL
LIN {X 0,Y 18.174,Z 592.41,A -85,B 0,C 180,E1 -32001.048,E2 -32001.048} C_VEL
LIN {X 0,Y 22.101,Z 587.911,A -85,B 0,C 180,E1 -32010.23,E2 -32010.23} C_VEL
LIN {X 0,Y 24.752,Z 584.854,A -85,B 0,C 180,E1 -32011.79,E2 -32011.79} C_VEL
LIN {X 0,Y 25.753,Z 583.754,A -85,B 0,C 180,E1 -32011.721,E2 -32011.721} C_VEL
LIN {X 0,Y 26.621,Z 582.468,A -85,B 0,C 180,E1 -32016.186,E2 -32016.186} C_VEL
LIN {X 0,Y 26.911,Z 582.002,A -85,B 0,C 180,E1 -32024.86,E2 -32024.86} C_VEL
LIN {X 0,Y 26.993,Z 582.155,A -85,B 0,C 180,E1 -32029.528,E2 -32029.528} C_VEL
LIN {X 0,Y 25.652,Z 583.961,A -85,B 0,C 180,E1 -32032.779,E2 -32032.779} C_VEL
LIN {X 0,Y 22.815,Z 587.173,A -85,B 0,C 180,E1 -32033.739,E2 -32033.739} C_VEL
LIN {X 0,Y 14.148,Z 595.333,A -85,B 0,C 180,E1 -32033.345,E2 -32033.345} C_VEL
LIN {X 0,Y 7.092,Z 600.684,A -85,B 0,C 180,E1 -32032.101,E2 -32032.101} C_VEL
LIN {X 0,Y 5.722,Z 601.499,A -85,B 0,C 180,E1 -32019.025,E2 -32019.025} C_VEL
LIN {X 0,Y 15.88,Z 593.691,A -85,B 0,C 180,E1 -32012.242,E2 -32012.242} C_VEL
LIN {X 0,Y 23.908,Z 585.782,A -85,B 0,C 180,E1 -32011.851,E2 -32011.851} C_VEL
LIN {X 0,Y 24.752,Z 584.854,A -85,B 0,C 180,E1 -32011.79,E2 -32011.79} C_VEL
LIN {X 0,Y 28.23,Z 586.2,A -85,B 0,C 180,E1 -32011.576,E2 -32011.576} C_VEL
LIN {X 0,Y 28.23,Z 600,A -85,B 0,C 180,E1 -32011.576,E2 -32011.576} C_VEL
LIN {X 0,Y 28.23,Z 600,A -85,B 0,C 180,E1 -32011.576,E2 -32011.576}

QRS_NEXT_CUT()

QRS_NEXT()
QRS_HOME()

END
